FUNCTION_BLOCK ABSTRACT FB_IOLinkDevice EXTENDS FB_BaseDevice
VAR_INPUT
    // This is presented as a linkable input in the main project via a GVL	
    PQIStatusInput AT %I* : BYTE;
END_VAR

END_FUNCTION_BLOCK

(* stored: Version 1.1.0.1, ProductVersion 3.1.4024.12
   POU FB_IOLinkDevice: Id {589e6482-7e3f-45cf-ba29-92bc74f578c6}, SpecialFunc None *)
